// TIA Portal project "compile_islemi_ve_hata_tamponu" (V18)

(* hardware
DEVICE "S7-1200 station_1"  S7-1200 Station
   slot 0: "Rack_0"  S7-1200 Rack  Rack  V1.0
   slot 1: "PLC_1"  CPU 1214C DC/DC/DC  6ES7 214-1AG40-0XB0  V4.6
*)

// ===== PLC "PLC_1"  CPU 1214C DC/DC/DC =====

VAR_GLOBAL   // PLC tag table "Default tag table"
   "Tag_1" AT %MW2 : Word;
   "Tag_2" AT %MW4 : UInt;
   "Tag_3" AT %MW6 : UInt;
   "Tag_4" AT %MW0 : Int;
END_VAR

ORGANIZATION_BLOCK "Main"   // OB1, LAD, ProgramCycle
TITLE = "Main Program Sweep (Cycle)"
{ S7_Optimized_Access := 'TRUE' }
VERSION : 0.1
   VAR_INPUT
      Initial_Call : Bool;   // Initial call of this OB
      Remanence : Bool;   // =True, if remanent data are available
   END_VAR
BEGIN

REGION Network 1
   // hatalı işlem varsa compile yapılır 
   // aşağıda uyarıyı görürürüz.
   // Yeşil oka tıkladığımız zaman bizi hatanın olduğu yere götürür. mavi markla işaretli yere gönderir
   // sarı uarı varsa error lambası yanıp söner
   // hatayı bulmak için online and diagnostic kısmına girilir ve diagnostic status tna hata durumu öğrenilir. Buffer kısmında hata nedeni görülebilir. Hatayı event kısmından kaydedebiliriz. Open editöre tıkladığımızda hataya gönderilir.
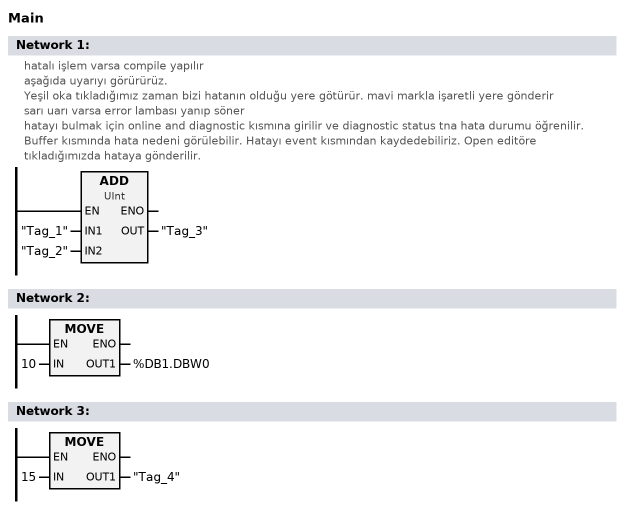
   RUNG wire#powerrail
      { S7_Templates := "SrcType := UInt" } Add(in1 := "Tag_1", in2 := "Tag_2", out => "Tag_3")
   END_RUNG
   // the same network as SCL:
   "Tag_3" := "Tag_1" + "Tag_2";
END_REGION

REGION Network 2
   RUNG wire#powerrail
      Move(in := 10, out1 => %DB1.DBW0)
   END_RUNG
   // the same network as SCL:
   %DB1.DBW0 := 10;
END_REGION

REGION Network 3
   RUNG wire#powerrail
      Move(in := 15, out1 => "Tag_4")
   END_RUNG
   // the same network as SCL:
   "Tag_4" := 15;
END_REGION
END_ORGANIZATION_BLOCK